// TIA Portal V17 export
// export: Created 2025-03-05T07:58:52.4060345Z, ExportSetting WithDefaults, DisplayName Totally Integrated Automation Portal, DisplayVersion V17 Update 8, DisplayName TIA Portal Openness, DisplayVersion V17 Update 8, DisplayName TIA Portal Version Control Interface, DisplayVersion V17, DisplayName SINAMICS Startdrive Advanced, DisplayVersion V17 SP2, DisplayName SINAMICS Startdrive G110M, G120, G120C, G120D, G120P, G115D, DisplayVersion V17 SP2, DisplayName SINAMICS Startdrive G130, G150, S120, S150, SINAMICS MV, S210, DisplayVersion V17 SP2, DisplayName STEP 7 Professional, DisplayVersion V17 Update 8, DisplayName SINUMERIK ONE STEP 7 Toolbox, DisplayVersion V17 Update 12, DisplayName SINUMERIK 840D sl STEP 7 Toolbox, DisplayVersion V17 Update 12, DisplayName STEP 7 Safety, DisplayVersion V17 Update 6, DisplayName WinCC Advanced, DisplayVersion V17 Update 8
DATA_BLOCK "LBP_MFuncDecListSignals"   // DB76
TITLE = M decoding acc. to list / Decodificación M seg. lista / M-Decodierung gem. Liste
{ S7_Optimized_Access := 'FALSE'; DB_Accessible_From_OPC_UA := 'FALSE' }
AUTHOR : SINUMERIK
FAMILY : SINUMERIK_ONE
VERSION : 6.15
// Interface between user program and NCK, contains the signal list for the request and acknowledgment of the M functions configured with LBP_MFuncDecListConfig [DB75] / Interfaz entre programa de usuario y NCK, contiene la lista de señales para la solicitud y confirmación de las funciones M configuradas con LBP_MFuncDecListConfig [DB75] / Schnittstelle zwischen Anwenderprogramm und NCK, enthält die Signalliste für die Anforderung und Quitteriung der mit LBP_MFuncDecListConfig [DB75] konfigurierten M-Funktionen
// stored: AutoNumber false, DBAccessibleFromOPCUA false, DBAccessibleFromWebserver true, IsOnlyStoredInLoadMemory false, IsWriteProtectedInAS false
   VAR
      MSigGrp1 : Struct
         MSig : Array[0..15] of Bool;
      END_STRUCT;
      MSigGrp2 : Struct
         MSig : Array[0..15] of Bool;
      END_STRUCT;
      MSigGrp3 : Struct
         MSig : Array[0..15] of Bool;
      END_STRUCT;
      MSigGrp4 : Struct
         MSig : Array[0..15] of Bool;
      END_STRUCT;
      MSigGrp5 : Struct
         MSig : Array[0..15] of Bool;
      END_STRUCT;
      MSigGrp6 : Struct
         MSig : Array[0..15] of Bool;
      END_STRUCT;
      MSigGrp7 : Struct
         MSig : Array[0..15] of Bool;
      END_STRUCT;
      MSigGrp8 : Struct
         MSig : Array[0..15] of Bool;
      END_STRUCT;
      MSigGrp9 : Struct
         MSig : Array[0..15] of Bool;
      END_STRUCT;
      MSigGrp10 : Struct
         MSig : Array[0..15] of Bool;
      END_STRUCT;
      MSigGrp11 : Struct
         MSig : Array[0..15] of Bool;
      END_STRUCT;
      MSigGrp12 : Struct
         MSig : Array[0..15] of Bool;
      END_STRUCT;
      MSigGrp13 : Struct
         MSig : Array[0..15] of Bool;
      END_STRUCT;
      MSigGrp14 : Struct
         MSig : Array[0..15] of Bool;
      END_STRUCT;
      MSigGrp15 : Struct
         MSig : Array[0..15] of Bool;
      END_STRUCT;
      MSigGrp16 : Struct
         MSig : Array[0..15] of Bool;
      END_STRUCT;
   END_VAR
BEGIN
END_DATA_BLOCK
